{attribute 'GeneratedUsingTerminal: EL6631-0000-0016'}
{attribute addProperty BoxType "EL6631-0000-0016"}
{attribute addProperty Id "InfoDataAT %I*InfoData_41C547A32"}
{attribute addProperty CRC "3204926373"}
{attribute addProperty Size "2"}
TYPE EL6631_BF074BA5 EXTENDS EtcSlaveTerminalBase_947E5A46 :
STRUCT
	{attribute addProperty Name "InfoData"}
	InfoData : InfoData_41C547A3;
END_STRUCT
END_TYPE

(* stored: Version 1.2.0.0, ProductVersion 3.1.4024.9
   DUT EL6631_BF074BA5: Id {d8bd4814-7692-4f1c-ba44-da74a6a7b3e1} *)
